Staubli VAL3: getDetectFrame.pgx

public program getDetectFrame(num x_nConvNum (dimensions=1), frame& x_fDetectFrame (dimensions=1), frame x_fRefFrame (dimensions=1), num& x_nError (dimensions=1))
begin
  // This program returns the position and orientation of the detection
  //  device frame in reference to the frame x_fRefFrame.
  //
  // Input Param
  //  x_nConvNum : Conveyor number
  //  x_fRefFrame: Reference frame from which the coordinates of
  //                x_fDetection should be returned.
  //
  // Output param
  //  x_fDetection: Coordinates of the detection device frame that have
  //                 been taught during calibration.
  //  x_nError    : Error code
  //    0    --> No error
  //    14   --> Conveyor library not started, the frame cannot be computed.
  //
  //----------------------------------------------------------------
  //
  switch x_nConvNum
    case 0
      if cnv0:libExist("getDetectFrame()")
        call cnv0:getDetectFrame(x_fDetectFrame,x_fRefFrame,x_nError)
      else
        nStatus=-1
      endIf
    break
    case 1
      if cnv1:libExist("getDetectFrame()")
        call cnv1:getDetectFrame(x_fDetectFrame,x_fRefFrame,x_nError)
      else
        nStatus=-1
      endIf
    break
  endSwitch
end
